FUNCTION F_normalization : LREAL
VAR_INPUT
	x : LREAL;
	mean : LREAL;
	std : LREAL;
END_VAR
VAR_OUTPUT
	x_nor : LREAL;
END_VAR

x_nor := (x - mean) / std;

END_FUNCTION

(* stored: Version 1.1.0.1, ProductVersion 3.1.4024.12
   POU F_normalization: Id {efbe80a6-deef-4140-83e9-ead59fb6ee0d}, SpecialFunc None *)
